// TIA Portal V20 export
TYPE "LER_typeMarkAndReadTrackingData"
// stored: Access Published
   STRUCT
      finished { ExternalWritable := 'False'} : Bool;
      result { ExternalWritable := 'False'} : Bool;
      data { ExternalWritable := 'False'} : String[32];
   END_STRUCT;
END_TYPE
